PROGRAM MAIN
VAR
	dataService : ADSDataService;
	newDataService : mqttCommsAdaptor;
	myMachine : MachineControl := (DataService := newDataService);
END_VAR

END_PROGRAM

(* stored: Version 1.1.0.1, ProductVersion 3.1.4024.12
   POU MAIN: Id {8df75bd0-3f8f-4732-b781-bc9d1ba921fd}, SpecialFunc None *)
